(* LS Electric XG5000 project: 11_02_4project *)
(* PLC LSPLC *)

PROGRAM NewProgram (* task: 스캔 프로그램 *)
VAR
    in1 : DWORD := 4860066;
    in2 : DWORD := 8710306;
    in3 : DWORD := 8988834;
    in4 : DWORD := 9048994;
    in5 : DWORD := 9053346;
    in6 : DWORD := 9054286;
    in7 : DWORD := 3811489;
    in8 : DWORD := 9054354;
    INST : TON;
    INST1 : TON;
    INST2 : TON;
    INST3 : TON;
    INST4 : TON;
    INST5 : TON;
    INST6 : TON;
    INST7 : TON;
END_VAR
VAR
    _e1 : R_TRIG;
    _e2 : R_TRIG;
    _e3 : R_TRIG;
    _e4 : R_TRIG;
    _e5 : R_TRIG;
    _e6 : R_TRIG;
    _e7 : R_TRIG;
    _e8 : R_TRIG;
END_VAR

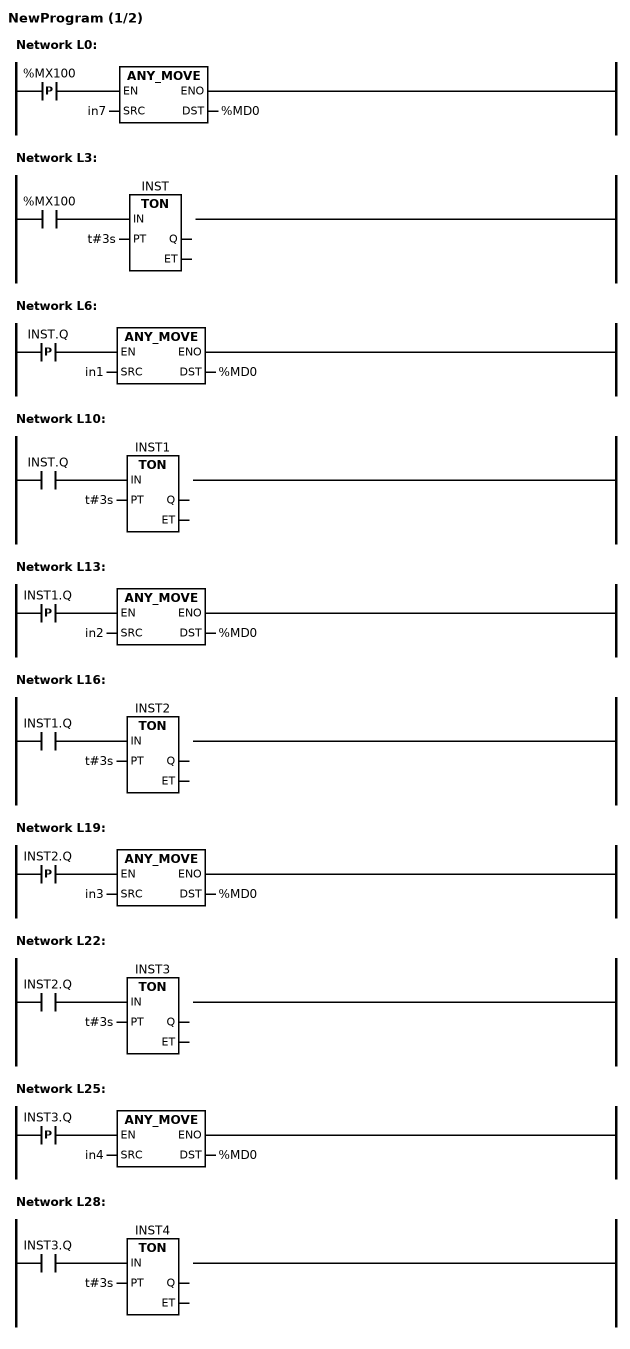
(* Rung L0 *)
_e1(CLK := %MX100);
IF _e1.Q THEN %MD0 := ANY_MOVE(SRC := in7); END_IF;
(* Rung L3 *)
INST(IN := %MX100, PT := t#3s);
(* Rung L6 *)
_e2(CLK := INST.Q);
IF _e2.Q THEN %MD0 := ANY_MOVE(SRC := in1); END_IF;
(* Rung L10 *)
INST1(IN := INST.Q, PT := t#3s);
(* Rung L13 *)
_e3(CLK := INST1.Q);
IF _e3.Q THEN %MD0 := ANY_MOVE(SRC := in2); END_IF;
(* Rung L16 *)
INST2(IN := INST1.Q, PT := t#3s);
(* Rung L19 *)
_e4(CLK := INST2.Q);
IF _e4.Q THEN %MD0 := ANY_MOVE(SRC := in3); END_IF;
(* Rung L22 *)
INST3(IN := INST2.Q, PT := t#3s);
(* Rung L25 *)
_e5(CLK := INST3.Q);
IF _e5.Q THEN %MD0 := ANY_MOVE(SRC := in4); END_IF;
(* Rung L28 *)
INST4(IN := INST3.Q, PT := t#3s);

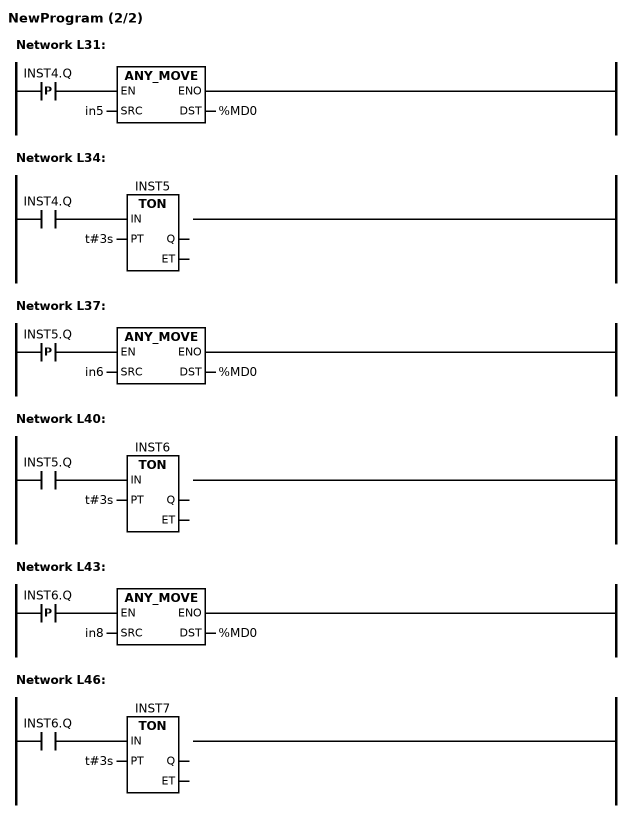
(* Rung L31 *)
_e6(CLK := INST4.Q);
IF _e6.Q THEN %MD0 := ANY_MOVE(SRC := in5); END_IF;
(* Rung L34 *)
INST5(IN := INST4.Q, PT := t#3s);
(* Rung L37 *)
_e7(CLK := INST5.Q);
IF _e7.Q THEN %MD0 := ANY_MOVE(SRC := in6); END_IF;
(* Rung L40 *)
INST6(IN := INST5.Q, PT := t#3s);
(* Rung L43 *)
_e8(CLK := INST6.Q);
IF _e8.Q THEN %MD0 := ANY_MOVE(SRC := in8); END_IF;
(* Rung L46 *)
INST7(IN := INST6.Q, PT := t#3s);
END_PROGRAM